// SIMATIC S7-200 SMART project (STEP 7-Micro/WIN SMART), CPU SR40

SYMBOL_TABLE 用户定义1
起动按钮             I0.0
已夹紧              I0.1
大孔钻完             I0.2
大钻升到位            I0.3
小孔钻完             I0.4
小钻升到位            I0.5
旋转到位             I0.6
已松开              I0.7
大钻升按钮            I1.0
大钻降按钮            I1.1
小钻升按钮            I1.2
小钻降按钮            I1.3
正转按钮             I1.4
反转按钮             I1.5
夹紧按钮             I1.6
松开按钮             I1.7
自动开关             I2.0
夹紧阀              Q0.0
大钻头降             Q0.1
大钻头升             Q0.2
小钻头降             Q0.3
小钻头升             Q0.4
工件正转             Q0.5
松开阀              Q0.6
工件反转             Q0.7
END_SYMBOL_TABLE

ORGANIZATION_BLOCK 主程序:OB1
TITLE=程序注释
BEGIN
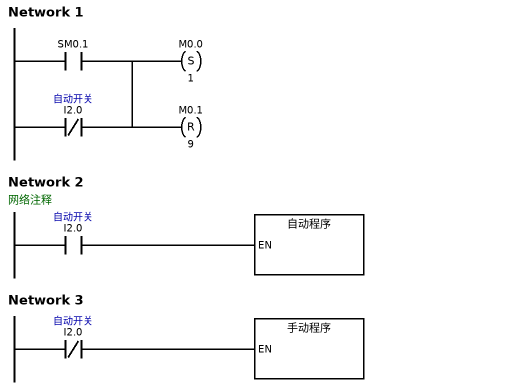
Network 1
LD     SM0.1
ON     自动开关:I2.0
S      M0.0, 1
R      M0.1, 9
Network 2
// 网络注释
LD     自动开关:I2.0
CALL   自动程序:SBR0
Network 3
LDN    自动开关:I2.0
CALL   手动程序:SBR1
END_ORGANIZATION_BLOCK

SUBROUTINE_BLOCK 自动程序:SBR0
TITLE=子程序注释
BEGIN
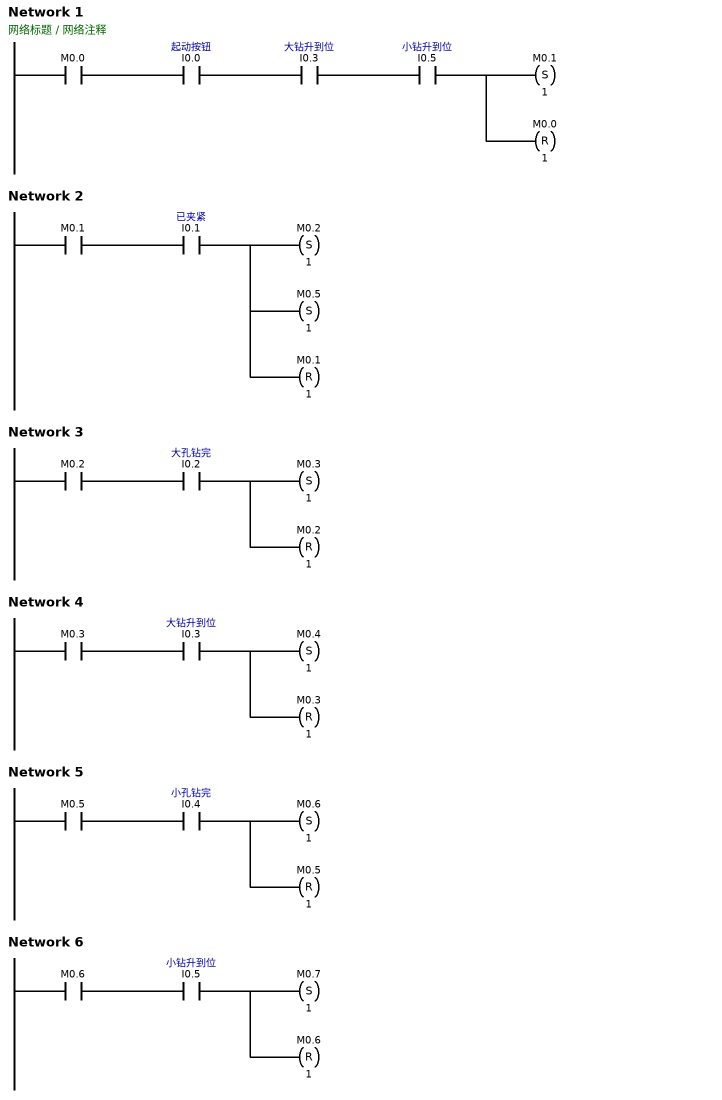
Network 1
// 网络标题
// 网络注释
LD     M0.0
A      起动按钮:I0.0
A      大钻升到位:I0.3
A      小钻升到位:I0.5
S      M0.1, 1
R      M0.0, 1
Network 2
LD     M0.1
A      已夹紧:I0.1
S      M0.2, 1
S      M0.5, 1
R      M0.1, 1
Network 3
LD     M0.2
A      大孔钻完:I0.2
S      M0.3, 1
R      M0.2, 1
Network 4
LD     M0.3
A      大钻升到位:I0.3
S      M0.4, 1
R      M0.3, 1
Network 5
LD     M0.5
A      小孔钻完:I0.4
S      M0.6, 1
R      M0.5, 1
Network 6
LD     M0.6
A      小钻升到位:I0.5
S      M0.7, 1
R      M0.6, 1
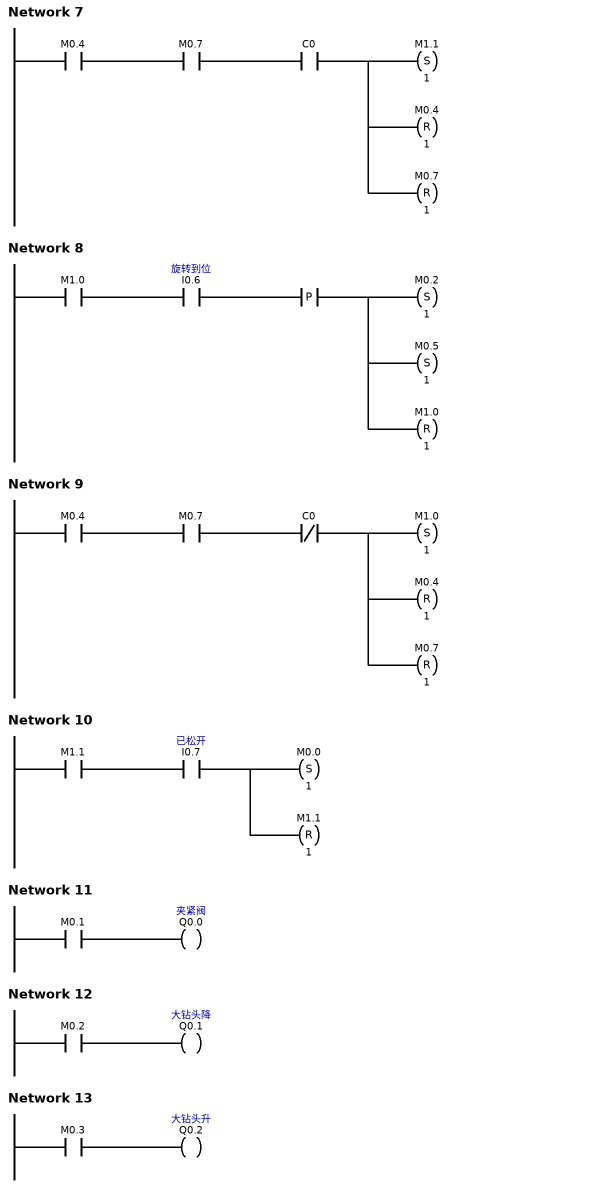
Network 7
LD     M0.4
A      M0.7
A      C0
S      M1.1, 1
R      M0.4, 1
R      M0.7, 1
Network 8
// (network saved uncompiled; LAD cells follow)
// row 0: c0 -| |- M1.0  c1 -| |- 旋转到位:I0.6  c2 -|P|-  v  c3 -(S) M0.2, 1
// row 1: c2 ^v  c3 -(S) M0.5, 1
// row 2: c2 ^  c3 -(R) M1.0, 1
Network 9
LD     M0.4
A      M0.7
AN     C0
S      M1.0, 1
R      M0.4, 1
R      M0.7, 1
Network 10
LD     M1.1
A      已松开:I0.7
S      M0.0, 1
R      M1.1, 1
Network 11
LD     M0.1
=      夹紧阀:Q0.0
Network 12
LD     M0.2
=      大钻头降:Q0.1
Network 13
LD     M0.3
=      大钻头升:Q0.2
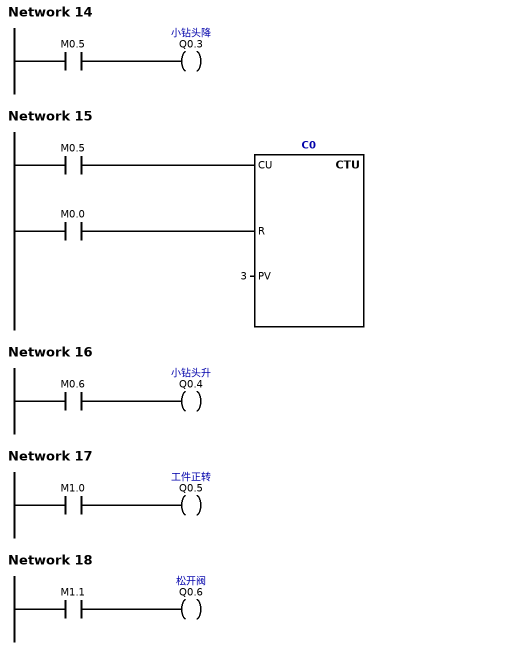
Network 14
LD     M0.5
=      小钻头降:Q0.3
Network 15
LD     M0.5
LD     M0.0
CTU    C0, 3
Network 16
LD     M0.6
=      小钻头升:Q0.4
Network 17
LD     M1.0
=      工件正转:Q0.5
Network 18
LD     M1.1
=      松开阀:Q0.6
END_SUBROUTINE_BLOCK

SUBROUTINE_BLOCK 手动程序:SBR1
TITLE=子程序注释
BEGIN
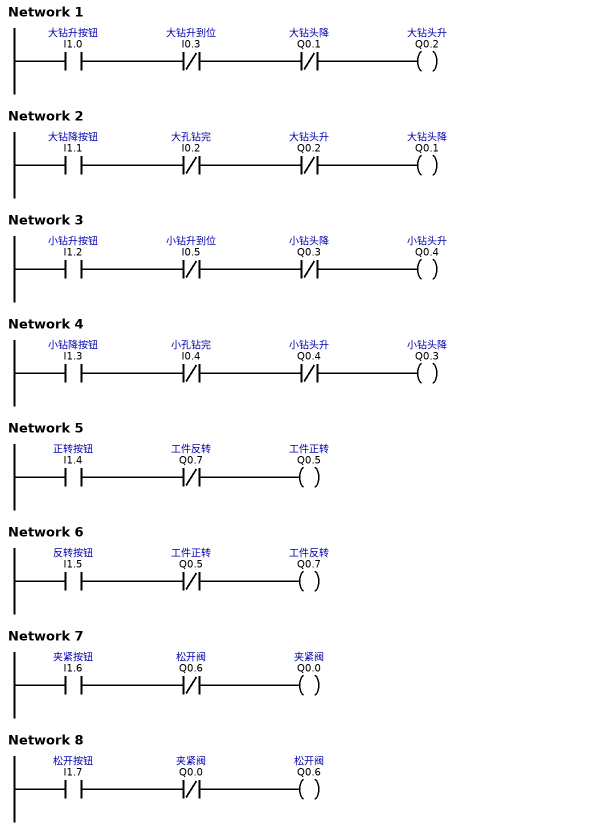
Network 1
LD     大钻升按钮:I1.0
AN     大钻升到位:I0.3
AN     大钻头降:Q0.1
=      大钻头升:Q0.2
Network 2
LD     大钻降按钮:I1.1
AN     大孔钻完:I0.2
AN     大钻头升:Q0.2
=      大钻头降:Q0.1
Network 3
LD     小钻升按钮:I1.2
AN     小钻升到位:I0.5
AN     小钻头降:Q0.3
=      小钻头升:Q0.4
Network 4
LD     小钻降按钮:I1.3
AN     小孔钻完:I0.4
AN     小钻头升:Q0.4
=      小钻头降:Q0.3
Network 5
LD     正转按钮:I1.4
AN     工件反转:Q0.7
=      工件正转:Q0.5
Network 6
LD     反转按钮:I1.5
AN     工件正转:Q0.5
=      工件反转:Q0.7
Network 7
LD     夹紧按钮:I1.6
AN     松开阀:Q0.6
=      夹紧阀:Q0.0
Network 8
LD     松开按钮:I1.7
AN     夹紧阀:Q0.0
=      松开阀:Q0.6
END_SUBROUTINE_BLOCK
